// TwinCAT 3 PLC project PLC1
// ProgramVersion: 3.1.4024.0
// libraries:
//   Tc2_Standard, * (Beckhoff Automation GmbH)
//   Tc2_System, * (Beckhoff Automation GmbH)
//   Tc3_Module, * (Beckhoff Automation GmbH)
// project tree:
//   / PlcTask.TcTTO
//   POUs/ main.TcPOU

CONFIGURATION PLC1
    RESOURCE PLC ON TwinCAT3
        TASK PlcTask(INTERVAL := T#10ms, PRIORITY := 20);
        PROGRAM main WITH PlcTask : main;
    END_RESOURCE
END_CONFIGURATION

// ---- POUs/main.TcPOU
PROGRAM main
VAR
	//sensori
	SensoreStart : BOOL := FALSE;
	SensoreReset : BOOL := FALSE;
	SensoreFCBottom : BOOL := FALSE;
	SensoreFCTop : BOOL := FALSE;
	SensoreFCS : BOOL := FALSE;
	SensoreFCD : BOOL := FALSE;
	SensoreFCP : BOOL := FALSE;
	SensoreGrasp : BOOL := FALSE;
	SensoreRelease : BOOL := FALSE;
	SensoreRulloOccupato : BOOL := FALSE;
	SensoreVascaVuota : BOOL := FALSE;
	{attribute 'OPC.UA.DA' := '1'}
	SensoreIsGiorno : BOOL := FALSE;
	SensoreSerbatoioOn : BOOL := FALSE;
	SensoreSerbatoioFull : BOOL := TRUE;
	SensoreSerbatoioEmpty : BOOL := FALSE;
	SensoreCondizionatore : BOOL := FALSE;
	SensoreApriFinestra : BOOL := FALSE;
	SensoreTempCalda : BOOL := FALSE;
	SensoreTempFredda : BOOL := FALSE;
	SensoreO2Low : BOOL := FALSE;
	SensorePianta1Pronta : BOOL := FALSE;
	SensorePianta2Pronta : BOOL := FALSE;
	//attuatori
	AttuatBraccioGiu : BOOL := FALSE;
	AttuatBraccioSu : BOOL := FALSE;
	AttuatBraccioSx : BOOL := FALSE;
	AttuatBraccioDx : BOOL := FALSE;
	AttuatBraccioPresa : BOOL := FALSE;
	AttuatBraccioRilascio : BOOL := FALSE;
	AttuatRiempiSerbatoio : BOOL := FALSE;
	AttuatSvuotaSerbatoio : BOOL := FALSE;
	AttuatFinestra : BOOL := FALSE;
	AttuatCondizionatore : BOOL := FALSE;
	AttuatRullo : BOOL := FALSE;
	AttuatLampada : BOOL := FALSE;
	
	//WatchDog e Allarme
	WatchDog : TON;
	TimerWatchDog : TIME := TIME#10S;
	{attribute 'OPC.UA.DA' := '1'}
	Allarme1 : BOOL := FALSE;
	{attribute 'OPC.UA.DA' := '1'}
	ContatorePiante : INT := 0;
	
	//Variabili RunTime per SCADA
	{attribute 'OPC.UA.DA' := '1'}
	Temperatura : LREAL;
	{attribute 'OPC.UA.DA' := '1'}
	Ossigeno: LREAL;
	
	AggiuntoPianta : BOOL := FALSE;
END_VAR

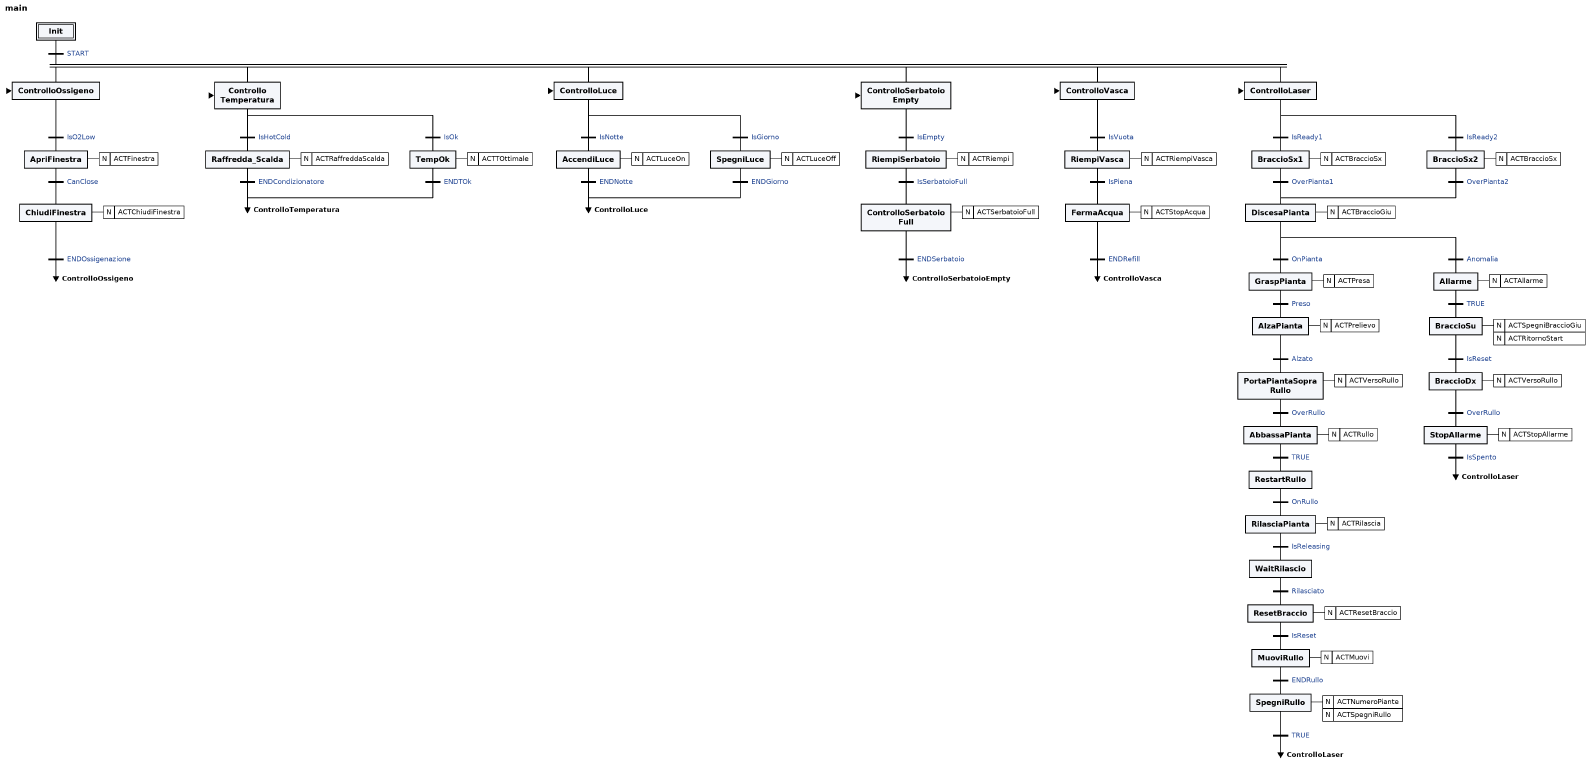
INITIAL_STEP Init:
END_STEP
TRANSITION FROM Init TO (ControlloOssigeno, ControlloTemperatura, ControlloLuce, ControlloSerbatoioEmpty, ControlloVasca, ControlloLaser)
    := START;
END_TRANSITION
STEP ControlloOssigeno:
END_STEP
TRANSITION FROM ControlloOssigeno TO ApriFinestra
    := IsO2Low;
END_TRANSITION
STEP ApriFinestra:
    ACTFinestra(N);
END_STEP
TRANSITION FROM ApriFinestra TO ChiudiFinestra
    := CanClose;
END_TRANSITION
STEP ChiudiFinestra:
    ACTChiudiFinestra(N);
END_STEP
TRANSITION FROM ChiudiFinestra TO ControlloOssigeno
    := ENDOssigenazione;
END_TRANSITION
STEP ControlloTemperatura:
END_STEP
TRANSITION FROM ControlloTemperatura TO Raffredda_Scalda
    := IsHotCold;
END_TRANSITION
STEP Raffredda_Scalda:
    ACTRaffreddaScalda(N);
END_STEP
TRANSITION FROM Raffredda_Scalda TO ControlloTemperatura
    := ENDCondizionatore;
END_TRANSITION
TRANSITION FROM ControlloTemperatura TO TempOk
    := IsOk;
END_TRANSITION
STEP TempOk:
    ACTTOttimale(N);
END_STEP
TRANSITION FROM TempOk TO ControlloTemperatura
    := ENDTOk;
END_TRANSITION
STEP ControlloLuce:
END_STEP
TRANSITION FROM ControlloLuce TO AccendiLuce
    := IsNotte;
END_TRANSITION
STEP AccendiLuce:
    ACTLuceOn(N);
END_STEP
TRANSITION FROM AccendiLuce TO ControlloLuce
    := ENDNotte;
END_TRANSITION
TRANSITION FROM ControlloLuce TO SpegniLuce
    := IsGiorno;
END_TRANSITION
STEP SpegniLuce:
    ACTLuceOff(N);
END_STEP
TRANSITION FROM SpegniLuce TO ControlloLuce
    := ENDGiorno;
END_TRANSITION
STEP ControlloSerbatoioEmpty:
END_STEP
TRANSITION FROM ControlloSerbatoioEmpty TO RiempiSerbatoio
    := IsEmpty;
END_TRANSITION
STEP RiempiSerbatoio:
    ACTRiempi(N);
END_STEP
TRANSITION FROM RiempiSerbatoio TO ControlloSerbatoioFull
    := IsSerbatoioFull;
END_TRANSITION
STEP ControlloSerbatoioFull:
    ACTSerbatoioFull(N);
END_STEP
TRANSITION FROM ControlloSerbatoioFull TO ControlloSerbatoioEmpty
    := ENDSerbatoio;
END_TRANSITION
STEP ControlloVasca:
END_STEP
TRANSITION FROM ControlloVasca TO RiempiVasca
    := IsVuota;
END_TRANSITION
STEP RiempiVasca:
    ACTRiempiVasca(N);
END_STEP
TRANSITION FROM RiempiVasca TO FermaAcqua
    := IsPiena;
END_TRANSITION
STEP FermaAcqua:
    ACTStopAcqua(N);
END_STEP
TRANSITION FROM FermaAcqua TO ControlloVasca
    := ENDRefill;
END_TRANSITION
STEP ControlloLaser:
END_STEP
TRANSITION FROM ControlloLaser TO BraccioSx1
    := IsReady1;
END_TRANSITION
STEP BraccioSx1:
    ACTBraccioSx(N);
END_STEP
TRANSITION FROM BraccioSx1 TO DiscesaPianta
    := OverPianta1;
END_TRANSITION
TRANSITION FROM ControlloLaser TO BraccioSx2
    := IsReady2;
END_TRANSITION
STEP BraccioSx2:
    ACTBraccioSx(N);
END_STEP
TRANSITION FROM BraccioSx2 TO DiscesaPianta
    := OverPianta2;
END_TRANSITION
STEP DiscesaPianta:
    ACTBraccioGiu(N);
END_STEP
TRANSITION FROM DiscesaPianta TO GraspPianta
    := OnPianta;
END_TRANSITION
STEP GraspPianta:
    ACTPresa(N);
END_STEP
TRANSITION FROM GraspPianta TO AlzaPianta
    := Preso;
END_TRANSITION
TRANSITION FROM DiscesaPianta TO Allarme
    := Anomalia;
END_TRANSITION
STEP Allarme:
    ACTAllarme(N);
END_STEP
TRANSITION FROM Allarme TO BraccioSu
    := TRUE;
END_TRANSITION
STEP BraccioSu:
    ACTSpegniBraccioGiu(N);
    ACTRitornoStart(N);
END_STEP
TRANSITION FROM BraccioSu TO BraccioDx
    := IsReset;
END_TRANSITION
STEP BraccioDx:
    ACTVersoRullo(N);
END_STEP
TRANSITION FROM BraccioDx TO StopAllarme
    := OverRullo;
END_TRANSITION
STEP StopAllarme:
    ACTStopAllarme(N);
END_STEP
TRANSITION FROM StopAllarme TO ControlloLaser
    := IsSpento;
END_TRANSITION
STEP AlzaPianta:
    ACTPrelievo(N);
END_STEP
TRANSITION FROM AlzaPianta TO PortaPiantaSopraRullo
    := Alzato;
END_TRANSITION
STEP PortaPiantaSopraRullo:
    ACTVersoRullo(N);
END_STEP
TRANSITION FROM PortaPiantaSopraRullo TO AbbassaPianta
    := OverRullo;
END_TRANSITION
STEP AbbassaPianta:
    ACTRullo(N);
END_STEP
TRANSITION FROM AbbassaPianta TO RestartRullo
    := TRUE;
END_TRANSITION
STEP RestartRullo:
END_STEP
TRANSITION FROM RestartRullo TO RilasciaPianta
    := OnRullo;
END_TRANSITION
STEP RilasciaPianta:
    ACTRilascia(N);
END_STEP
TRANSITION FROM RilasciaPianta TO WaitRilascio
    := IsReleasing;
END_TRANSITION
STEP WaitRilascio:
END_STEP
TRANSITION FROM WaitRilascio TO ResetBraccio
    := Rilasciato;
END_TRANSITION
STEP ResetBraccio:
    ACTResetBraccio(N);
END_STEP
TRANSITION FROM ResetBraccio TO MuoviRullo
    := IsReset;
END_TRANSITION
STEP MuoviRullo:
    ACTMuovi(N);
END_STEP
TRANSITION FROM MuoviRullo TO SpegniRullo
    := ENDRullo;
END_TRANSITION
STEP SpegniRullo:
    ACTNumeroPiante(N);
    ACTSpegniRullo(N);
END_STEP
TRANSITION FROM SpegniRullo TO ControlloLaser
    := TRUE;
END_TRANSITION

ACTION ACTAllarme:
Allarme1 := TRUE;
END_ACTION

ACTION ACTBraccioGiu:
AttuatBraccioSx := FALSE;
AttuatBraccioGiu := TRUE;
WatchDog(IN := TRUE, PT := TimerWatchDog);
END_ACTION

ACTION ACTBraccioSx:
AttuatBraccioSx := TRUE;
END_ACTION

ACTION ACTChiudiFinestra:
AttuatFinestra := FALSE;
END_ACTION

ACTION ACTFinestra:
AttuatFinestra := TRUE;
END_ACTION

ACTION ACTLuceOff:
AttuatLampada := FALSE;
END_ACTION

ACTION ACTLuceOn:
AttuatLampada := TRUE;
END_ACTION

ACTION ACTMuovi:
AttuatBraccioSu := FALSE;
AttuatRullo := TRUE;
END_ACTION

ACTION ACTNumeroPiante:
IF AggiuntoPianta = FALSE THEN
	ContatorePiante := ContatorePiante+1;
	AggiuntoPianta := TRUE;
END_IF
END_ACTION

ACTION ACTPrelievo:
AttuatBraccioPresa := FALSE;
AttuatBraccioSu := TRUE;
END_ACTION

ACTION ACTPresa:
AttuatBraccioGiu := FALSE;
AttuatBraccioPresa := TRUE;
WatchDog(IN := FALSE, PT := TimerWatchDog);
AggiuntoPianta := FALSE;
END_ACTION

ACTION ACTRaffreddaScalda:
//Dovrebbe azionare il condizionare freddo
AttuatCondizionatore := TRUE;
END_ACTION

ACTION ACTResetBraccio:
AttuatBraccioRilascio := FALSE;
AttuatBraccioSu := TRUE;
END_ACTION

ACTION ACTRiempi:
AttuatRiempiSerbatoio := TRUE;
END_ACTION

ACTION ACTRiempiVasca:
AttuatSvuotaSerbatoio := TRUE;
END_ACTION

ACTION ACTRilascia:
AttuatBraccioGiu := FALSE;
AttuatBraccioRilascio := TRUE;
END_ACTION

ACTION ACTRitornoStart:
AttuatBraccioSu := TRUE;
END_ACTION

ACTION ACTRullo:
AttuatBraccioDx := FALSE;
AttuatBracciogiu := TRUE;
END_ACTION

ACTION ACTSerbatoioFull:
AttuatRiempiSerbatoio := FALSE;
END_ACTION

ACTION ACTSpegniBraccioGiu:
AttuatBraccioGiu := FALSE;
END_ACTION

ACTION ACTSpegniRullo:
AttuatRullo := FALSE;
END_ACTION

ACTION ACTStopAcqua:
AttuatSvuotaSerbatoio := FALSE;
END_ACTION

ACTION ACTStopAllarme:
AttuatBraccioDx := FALSE;
Allarme1 := FALSE;
WatchDog(IN := FALSE, PT := TimerWatchDog);
END_ACTION

ACTION ACTTOttimale:
AttuatCondizionatore := FALSE;
END_ACTION

ACTION ACTVersoRullo:
//QUI PUOI MERGIARE
AttuatBraccioSu := FALSE;
AttuatBraccioDx := TRUE;
END_ACTION

TRANSITION Alzato:
SensoreFCTop = TRUE
END_TRANSITION

TRANSITION Anomalia:
WatchDog.Q = TRUE
END_TRANSITION

TRANSITION CanClose:
SensoreApriFinestra = FALSE AND SensoreO2Low = FALSE
END_TRANSITION

TRANSITION ENDCondizionatore:
AttuatCondizionatore = TRUE AND SensoreCondizionatore = TRUE
END_TRANSITION

TRANSITION ENDGiorno:
AttuatLampada = FALSE
END_TRANSITION

TRANSITION ENDNotte:
AttuatLampada = TRUE
END_TRANSITION

TRANSITION ENDOssigenazione:
AttuatFinestra = FALSE
END_TRANSITION

TRANSITION ENDRefill:
AttuatSvuotaSerbatoio = FALSE
END_TRANSITION

TRANSITION ENDRullo:
SensoreRulloOccupato = FALSE
END_TRANSITION

TRANSITION ENDSerbatoio:
AttuatRiempiSerbatoio = FALSE
END_TRANSITION

TRANSITION ENDTOk:
AttuatCondizionatore = FALSE AND SensoreCondizionatore = FALSE
END_TRANSITION

TRANSITION IsEmpty:
SensoreSerbatoioEmpty = TRUE
END_TRANSITION

TRANSITION IsGiorno:
SensoreIsGiorno = TRUE
END_TRANSITION

TRANSITION IsHotCold:
SensoreTempCalda = TRUE OR SensoreTempFredda = TRUE
END_TRANSITION

TRANSITION IsNotte:
SensoreIsGiorno = FALSE
END_TRANSITION

TRANSITION IsO2Low:
SensoreO2Low = TRUE AND SensoreApriFinestra = TRUE
END_TRANSITION

TRANSITION IsOk:
SensoreTempFredda = FALSE AND SensoreTempCalda = FALSE
END_TRANSITION

TRANSITION IsPiena:
SensoreSerbatoioOn = FALSE AND SensoreVascaVuota = FALSE
END_TRANSITION

TRANSITION IsReady1:
SensorePianta1Pronta = TRUE
END_TRANSITION

TRANSITION IsReady2:
SensorePianta2Pronta = TRUE
END_TRANSITION

TRANSITION IsReleasing:
SensoreRelease = TRUE
END_TRANSITION

TRANSITION IsReset:
SensoreFCTop = TRUE
END_TRANSITION

TRANSITION IsSerbatoioFull:
SensoreSerbatoioFull = TRUE
END_TRANSITION

TRANSITION IsSpento:
Allarme1 = FALSE
END_TRANSITION

TRANSITION IsVuota:
 //AND SensoreSerbatoioOn = TRUE
SensoreVascaVuota = TRUE AND SensoreSerbatoioEmpty = FALSE
END_TRANSITION

TRANSITION OnPianta:
SensoreFCBottom = TRUE AND WatchDog.Q = FALSE
END_TRANSITION

TRANSITION OnRullo:
SensoreFCBottom = TRUE AND SensoreRulloOccupato = TRUE
END_TRANSITION

TRANSITION OverPianta1:
SensoreFCS = TRUE
END_TRANSITION

TRANSITION OverPianta2:
SensoreFCP = TRUE
END_TRANSITION

TRANSITION OverRullo:
SensoreFCD = TRUE
END_TRANSITION

TRANSITION Preso:
SensoreGrasp = TRUE
END_TRANSITION

TRANSITION RESTART:
SensoreReset = TRUE
END_TRANSITION

TRANSITION Rilasciato:
SensoreRelease = FALSE
END_TRANSITION

TRANSITION START:
SensoreStart = TRUE AND SensoreFCTop= TRUE AND SensoreFCD = TRUE AND SensoreRulloOccupato = FALSE
END_TRANSITION

END_PROGRAM
